FUNCTION_BLOCK Ass_LoadPic IMPLEMENTS ITF_AutoStructCommand
VAR_INPUT
END_VAR
VAR_OUTPUT
END_VAR
VAR
	strText	:STRING;
	i	:INT;
	_bProcessScan,_bInitialScan		: BOOL;
	_bHalt , _bError,_bHaltPause	: BOOL;
	nStep,nInitiStep ,nNextStep 	: INT;
	fbHomeInside,fbHomeOutside		: MC_Home;
	fbMC_GearIn						: MC_GearIn;
	fbMC_GearOut					: MC_GearOut;
	fbMC_AbsLoad1,fbMC_AbsLoad2		: MC_MoveAbsolute;
	fbMC_Mode1	,fbMC_Mode2			:MC_MoveModulo;
	fbMC_INC1,fbMC_INC2	:MC_MoveRelative;
	_tmrT0,tmrStopper							: TON;
	temp:DWORD;
	bReady: BOOL;
END_VAR

IF NOT _bInitialScan AND NOT _bProcessScan  THEN
	fbHomeInside.Execute:=FALSE;
	fbHomeOutside.Execute:=FALSE;
END_IF


IF NOT _bInitialScan THEN
	nInitiStep	:= 0;
END_IF

_bInitialScan:=FALSE;



IF NOT _bProcessScan THEN
	nNextStep	:= 0;
	nStep		:= 0;
END_IF

_bProcessScan	:=FALSE;






fbHomeInside(Axis:= Axis_load1,Position:= Setting_Unload1_ORG_Offset*-1,bCalibrationCam:= NOT Sen_AxisLoad1ORG);
fbHomeOutside(Axis:= Axis_load2,Position:= Setting_Unload2_ORG_Offset*-1,bCalibrationCam:= NOT Sen_AxisLoad2ORG);

METHOD _Clearfb : BOOL
VAR_INPUT
END_VAR
	fbMC_GearIn(Master:=Axis_load1,Slave:=Axis_load2,Execute:=FALSE);
	fbMC_GearOut(Slave:=Axis_load2,Execute:=FALSE);
	fbHomeInside(Axis:= Axis_load1,bCalibrationCam:= FALSE,Execute:=FALSE);
	fbHomeOutside(Axis:= Axis_load2,bCalibrationCam:= FALSE,Execute:=FALSE);
	_tmrT0(IN:=FALSE);
	nInitiStep:=0;
END_METHOD

{warning 'add property implementation'}
PROPERTY Connect : STRING(50)
GET
CASE nStep OF
 10:
	Connect	:= 'Seal In';
20:
	Connect	:= 'LoadIng';
 25:
	Connect	:= 'Seal In';	
	ELSE	
	Connect	:= '';		
END_CASE
END_GET
SET
END_SET
END_PROPERTY

PROPERTY Error : BOOL
GET
Error := _bError;
END_GET
END_PROPERTY

METHOD ErrorClear : BOOL
_bError	:= FALSE;
END_METHOD

{warning 'add method implementation '}
METHOD FB_init : BOOL
VAR_INPUT
	(* if TRUE, the retain variables are initialized (warm start / cold start)*)
	bInitRetains	: BOOL;
	(* if TRUE, the instance afterwards gets moved into the copy code (online change)*)
	bInCopyCode	: BOOL;
END_VAR
END_METHOD

{warning 'add method implementation '}
METHOD HaltStepContiune : BOOL
END_METHOD

METHOD Initialization : BOOL
VAR_INPUT
	_Testmode	:BOOL;
END_VAR
VAR
	bConfig: BOOL;
END_VAR
_bInitialScan	:= TRUE;

CASE nInitiStep OF
	0:
		RB_CS_PickIO.cmd_bBoxInPos	:=FALSE;
		fbMC_AbsLoad1(Axis:= Axis_load1,Velocity:= 100,Execute:= FALSE);
		fbMC_AbsLoad2(Axis:= Axis_load2,Velocity:= 100,Execute:= FALSE);
		fbHomeInside.Execute:=FALSE;
		fbHomeOutside.Execute:=FALSE;
		fbMC_GearOut(Slave:= Axis_load2,Execute:=FALSE);
		_tmrT0(IN:=FALSE);
		Cyl_UnloadDef.qExtendCoil	:= FALSE;
		strText:='ORG : Initial ';
		IF AssRoller.Initialization() THEN
			nInitiStep := 1;
		END_IF
	1:
		_tmrT0(IN:= NOT _tmrT0.Q ,PT:= T#1S);
		CASE Axis_load1.Status.MotionState OF
			MC_AXISSTATE_DISABLED:
			 	Axis_load1.ServoOn();
			MC_AXISSTATE_ERRORSTOP:
				Axis_load1.Reset();
			MC_AXISSTATE_STOPPING:
				Axis_load1.Stop();
			MC_AXISSTATE_SYNCHRONIZEDMOTION:
			;
		END_CASE;		
		CASE Axis_load2.Status.MotionState OF
			MC_AXISSTATE_DISABLED:
			 	Axis_load2.ServoOn();
			MC_AXISSTATE_ERRORSTOP:
				Axis_load2.Reset();
			MC_AXISSTATE_STOPPING:
				Axis_load2.Stop();
			MC_AXISSTATE_SYNCHRONIZEDMOTION:
				fbMC_GearOut(Slave:= Axis_load2,Execute:=TRUE);
		END_CASE;			
		
		IF  Axis_load1.Status.MotionState=MC_AXISSTATE_STANDSTILL AND Axis_load2.Status.MotionState=MC_AXISSTATE_STANDSTILL THEN
			_tmrT0(IN:=FALSE);
			nInitiStep	:=5 ;
		END_IF
		IF _tmrT0.Q THEN
			_tmrT0(IN:=FALSE);
			nInitiStep	:= 5;		
		END_IF
	5:
		bConfig			:=TRUE;
		IF NOT Axis_load1.Status.StandStill THEN
			bConfig			:=FALSE;
			EventLogger.eEventType		:= 4;
			EventLogger.strEventText	:= 'RightAxis Error ';	
			EventLogger();					
		END_IF
		IF NOT Axis_load2.Status.StandStill THEN
			bConfig			:=FALSE;
			EventLogger.eEventType		:= 4;
			EventLogger.strEventText	:= 'LefthtAxis Error';	
			EventLogger();					
		END_IF
		
		IF bConfig THEN
			IF NOT OP.xAutoMode THEN
				EventLogger.eEventType		:= 2;
				EventLogger.strEventText	:= 'LoadIn servo ORG Runing ';	
				EventLogger();
			END_IF;
			_tmrT0(IN:= FALSE);
			nInitiStep:= 10 ;
			strText:='ORG : Runing ';
			ELSE
			EventLogger.eEventType		:= 4;
			EventLogger.strEventText	:= 'Exceptions Cause interruptions!! ';	
			EventLogger();
			OP.xAutoRuning	:=FALSE;
			nInitiStep := nInitiStep +100;	
			strText:='ORG : Failed  ';
		END_IF			
		
	10:
		fbHomeInside.Execute:=TRUE;
		fbHomeOutside.Execute:=TRUE;
		fbMC_AbsLoad1(Axis:= Axis_load1,Position:= 0,Velocity:= RunParameter.Load_Velo,Execute:= fbHomeInside.Done );
		fbMC_AbsLoad2(Axis:= Axis_load2,Position:= 0,Velocity:= RunParameter.Load_Velo,Execute:=  fbHomeOutside.Done);
	
		IF fbMC_AbsLoad1.Done AND fbMC_AbsLoad2.Done THEN
			fbHomeInside.Execute:=FALSE;
			fbHomeOutside.Execute:=FALSE;
			fbMC_AbsLoad1(Axis:= Axis_load1,Velocity:= RunParameter.Load_Velo,Execute:=FALSE );
			fbMC_AbsLoad2(Axis:= Axis_load2,Velocity:= RunParameter.Load_Velo,Execute:=FALSE );
			strText:='ORG : Done ';
			nInitiStep	:= 20 ;
		END_IF
	20:
		Initialization := TRUE;

END_CASE;
END_METHOD

{warning 'add property implementation'}
PROPERTY NoEntry : BOOL
GET
END_GET
END_PROPERTY

{warning 'add method implementation '}
METHOD Pause : BOOL
END_METHOD

METHOD Process : BOOL
VAR_INPUT
	bHlatMode	: BOOL;
END_VAR
_bProcessScan	:= TRUE;
//判斷 

IF _bError THEN
	strText	:= 'OpenBox:Error ';
	strText	:= CONCAT(Status,INT_TO_STRING(nStep));
END_IF;
//半自動模式
IF NOT bHlatMode  THEN
	nStep:= nNextStep;	
END_IF;

_bHaltPause	:= nStep<> nNextStep;
IF _bError OR _bHaltPause THEN
	RETURN;
END_IF
fbMC_INC1(Axis:= Axis_load1,Distance:= 1005,Velocity:= RunParameter.Load_Velo);
fbMC_INC2(Axis:= Axis_load2,Distance:= 1005,Velocity:= RunParameter.Load_Velo);
fbMC_Mode1(Axis:= Axis_load1,Velocity:= fbMC_AbsLoad1.Velocity,Direction:= MC_Positive_Direction);
fbMC_Mode2(Axis:= Axis_load2,Velocity:= fbMC_AbsLoad1.Velocity,Direction:= MC_Positive_Direction);
fbMC_AbsLoad1(Axis:= Axis_load1,Position:= RunParameter.Load_RBLoadin,Velocity:= RunParameter.Load_Velo);
fbMC_AbsLoad2(Axis:= Axis_load2,Position:= RunParameter.Load_RBLoadin,Velocity:= RunParameter.Load_Velo);	

//主程序 
IF NOT _bHaltPause THEN
	CASE nStep OF
		0:
			fbMC_AbsLoad1.Execute:=FALSE;
			fbMC_AbsLoad2.Execute:=FALSE;
			fbMC_INC1.Execute:=FALSE;
			fbMC_INC2.Execute:= FALSE;
			fbMC_Mode1.Execute:= FALSE;
			fbMC_Mode2.Execute:= FALSE;
			fbHomeInside(Axis:= Axis_load1,Execute:=FALSE);
			fbHomeOutside(Axis:= Axis_load2,Execute:=FALSE);
			_tmrT0(IN:=FALSE);			
			nNextStep:= 5;
		
		5:
			fbMC_AbsLoad1(Axis:= Axis_load1,Position:= 0,Velocity:= RunParameter.Load_Velo,Execute:= TRUE);
			fbMC_AbsLoad2(Axis:= Axis_load2,Position:= 0,Velocity:= RunParameter.Load_Velo,Execute:= TRUE);		
			IF fbMC_AbsLoad1.Done AND fbMC_AbsLoad2.Done THEN
				fbMC_AbsLoad1(Axis:= Axis_load1,Velocity:= RunParameter.Load_Velo,Execute:=FALSE );
				fbMC_AbsLoad2(Axis:= Axis_load2,Velocity:= RunParameter.Load_Velo,Execute:=FALSE );
				nNextStep	:= 10 ;
			END_IF		
		10:
			IF OP.xAutoMode THEN
				IF M_Sealing2.Connect='LoadPic In' THEN	
					nNextStep	:= 11 ;
				END_IF;
			END_IF
			
			IF NOT OP.xAutoMode THEN
				IF Sen_BeltLoadOut THEN
					nNextStep	:= 11 ;
				END_IF;			
			END_IF

		11:
			_tmrT0(IN:= NOT Sen_BeltLoadOut ,pt:= T#0.5S);
			IF _tmrT0.Q THEN
				_tmrT0(IN:=FALSE);
				nNextStep	:= 15 ;
			END_IF
			
		15:
			Cyl_UnloadDef.qExtendCoil	:= TRUE;
			fbMC_Mode1.Execute:= TRUE;
			fbMC_Mode1.Position	:= Parameter_PERSISTENT.RunParameter.Load_RBLoadin;
			fbMC_Mode2.Execute:= TRUE;
			fbMC_Mode2.Position	:= Parameter_PERSISTENT.RunParameter.Load_RBLoadin;	
			IF fbMC_Mode1.Done AND fbMC_Mode2.Done THEN
				fbMC_Mode1.Execute:= FALSE;
				fbMC_Mode2.Execute:= FALSE;	
				nNextStep	:= 16 ;			
			END_IF


	
		16:
			IF Cyl_UnloadDef.iEndSensor  THEN
				nNextStep	:= 20 ;
			END_IF	
			
		20:	// 允許手臂loadin
			IF RB_CS.LoadingDone() THEN
				bReady	:= M_Sealing2.Connect = 'Ready';
				_tmrT0(IN:=FALSE);
				nNextStep	:= 25 ;
			END_IF	
		25:
			Cyl_UnloadDef.qExtendCoil	:= FALSE;
			IF Roller_LoadcellUD.iLowPos AND Cyl_UnloadDef.iOriginSensor THEN
				IF bReady THEN
					nNextStep	:= 30 ;
					ELSE
					nNextStep	:= 31 ;
				END_IF;	
			END_IF
		30:	
			tmrStopper(IN:= NOT Sen_UnloadLoadPos ,PT := T#0.5S);
			IF tmrStopper.q THEN
				Cyl_UnloadDef.qExtendCoil	:= TRUE;
			END_IF
			fbMC_INC1.Execute:= TRUE;
			fbMC_INC2.Execute:= TRUE;	
			IF fbMC_INC2.Done AND fbMC_INC1.Done THEN
				fbMC_INC1.Execute:= FALSE;
				fbMC_INC2.Execute:= FALSE;	
				bReady	:=FALSE;
				Cyl_UnloadDef.qExtendCoil	:= TRUE;
				tmrStopper(IN:=FALSE);
				nNextStep	:= 16 ;
			END_IF;
		31:	
			fbMC_Mode1.Execute:= TRUE;
			fbMC_Mode1.Position	:= 0;
			fbMC_Mode2.Execute:= TRUE;
			fbMC_Mode2.Position	:= 0;	
			IF fbMC_Mode1.Done AND fbMC_Mode2.Done THEN
				fbMC_Mode1.Execute:= FALSE;
				fbMC_Mode2.Execute:= FALSE;	
				nNextStep	:= 10 ;			
			END_IF
			
			(*
			IF Initialization(FALSE) THEN
				nNextStep	:= 0 ;
				IF bReady THEN
					nNextStep	:= 15 ;
				END_IF
			END_IF
		*)
		
			
		
	END_CASE;
END_IF;
		
Process	:= nStep =50;
END_METHOD

PROPERTY Status : STRING(50)
GET
END_GET
END_PROPERTY

END_FUNCTION_BLOCK

(* stored: Version 1.1.0.1, ProductVersion 3.1.4026.18
   POU Ass_LoadPic: Id {41058aa1-f0d8-4eea-8392-b9cb2c6e1dc2}, SpecialFunc None
   Method _Clearfb: Id {aad993d0-491f-4baf-a2f6-4ec83f321454}
   Property Connect: Id {dd733115-1bb2-4f8e-bc53-dbef49f5e4af}
   Get Get: Id {019cfa34-437d-40b0-9773-6999e0db6284}
   Set Set: Id {e35af6d6-9509-4a31-8e28-168b58415986}
   Property Error: Id {fe8e8953-d44b-430e-9c1e-c530422ebf25}
   Get Get: Id {1b99a44c-f662-40f2-9427-9b26fd181fb8}
   Method ErrorClear: Id {d8421e47-9747-4b75-8f39-7f46711a51da}
   Method FB_init: Id {3c67647f-4069-4f92-affe-311c7be04a50}
   Method HaltStepContiune: Id {ef121d40-ba23-4ebf-abc0-02af33e485ba}
   Method Initialization: Id {105550df-bf40-45a4-afe8-08ca51d11f31}
   Property NoEntry: Id {8ec65748-586b-4750-9ce0-856e1544908c}
   Get Get: Id {11ed35a8-a5c5-40d1-8ef2-a6a43ee5c9d3}
   Method Pause: Id {1c396a50-1f9f-419e-87a9-cb9845eeb508}
   Method Process: Id {a69da40f-2129-4cc7-975f-fe74944e7f4d}
   Property Status: Id {15589aae-c7ea-459f-af14-8a5808d9a3c9}
   Get Get: Id {9224472d-2189-4887-95ae-35748dfdad8b} *)
